(* CODESYS project Single_Axis_180501.export

Project tree, tasks and I/O mapping:
  program SingleAxis [ST]
*)

// SingleAxis
PROGRAM SingleAxis  // define a program, which realize the movement of one axis in both pos and neg direction.
VAR
	Enable : BOOL;
	StartMov : BOOL;
	MovAxis : INT := 0;
	FirstPos : REAL := -180; // negative direction with a value of 180
	SecondPos : REAL := 180;
	CurrentPos : REAL;
	Vel : REAL := 180;
	Acc : REAL := 180;
	Jerk : REAL := 180;
	stopTime : TIME := T#1S; // time = 1 s
	MovErr : BOOL;
	
	PowBlk : ArcaLibrary.MC_Power;// call the function block ( Poweron/-off) in the Arc_Lib.
	PowDone, PowErr : BOOL;
	
	MovState : INT;
	FirMov : ArcaLibrary.MC_MoveAbsolute; // the function block (Move)
	SecMov : ArcaLibrary.MC_MoveAbsolute;
	StopMov : ArcaLibrary.MC_Stop;
	dis_trig : r_trig; // trigger
	
	ReadPos : ArcaLibrary.MCAT_ReadAxisMeasures;
	StopTimer : ton; // timer
END_VAR

// in the beginning, enable the axis and set status PowerOn
PowBlk(Axis := MovAxis, Enable:=Enable, EnablePositive:=TRUE, EnableNegative:=TRUE, Status=>PowDone, Error=>PowErr); 
// read the axis position
ReadPos(axis := MovAxis, enable := PowBlk.Status, pos=> currentPos);
// set the trigger in false
dis_trig(clk := NOT startMov);
StopMov(axis := MovAxis, execute := dis_trig.Q, Deceleration := acc*10, jerk := jerk*10); // if trigger is true, stop the movement. In that moment, tigger is false

IF MovState > 20 AND NOT startMov THEN
	MovState := 20;    // if startMov is set to false, reset the machine state to 20
END_IF
CASE MovState OF // define different machine state
	0:
		IF PowDone THEN // check PowerOn
			MovState := 10;
		END_IF
	10:
		IF startMov THEN // check startMov
			MovState := 20;
		END_IF
	20:  //set the axis value to the function block without movement
		FirMov(axis := MovAxis, Execute := FALSE);
		SecMov(axis := MovAxis, Execute := FALSE);
		IF startMov THEN
			StopTimer(in:= FALSE); // if startMov is true, unuse the stop function
			MovState := 30;
		ELSE
			MovState := 0; // if startMov is false, back to begin
		END_IF
	30:  // command, then begin the first movement towards neg direction with 180 degree
		FirMov(axis := MovAxis, Execute := TRUE, Position := FirstPos   
			, Velocity := vel, Acceleration := acc, Deceleration := Acc, jerk := jerk
			, Direction := mcShortestWay, BufferMode := mcAborting 
			, Error => MovErr);
		IF FirMov.Done THEN // after movement is done, check if a delay is needed
			IF stopTime > T#0S THEN   // if a delay exist, execute it
				StopTimer (in := TRUE, PT := stopTime);
				MovState := 35;
			ELSE  // if not, skip to next step
				MovState := 40;
			END_IF
		END_IF
	35: // execute the delay, if delay time is defined
		StopTimer (in := TRUE, PT := stopTime); // Timer:  Set IN to true, and after PT, the output Q will be true. It means, if Q is set to true, Pt time is already gone
		IF StopTimer.Q THEN
			StopTimer(in:= FALSE);
			MovState := 40;
		END_IF
	40:  // execute the second movement, axis rotates in pos direction with 180 degree
		SecMov(axis := MovAxis, Execute := TRUE, Position := SecondPos
			, Velocity := vel, Acceleration := acc, Deceleration := Acc, jerk := jerk
			, Direction := mcShortestWay, BufferMode := mcAborting 
			, Error => MovErr);
		IF SecMov.Done THEN // after the movement, check if a delay is needed
			StopTimer (in := TRUE, PT := stopTime);
			IF stopTime > T#0S THEN
				MovState := 45;
			ELSE // when not, restart the cycle with step 20
			MovState := 20;
			END_IF
		END_IF
	45: // execute the delay for second movement
		StopTimer (in := TRUE, PT := stopTime);
		IF StopTimer.Q THEN
			StopTimer(in:= FALSE);
			MovState := 20;
		END_IF
END_CASE

END_PROGRAM
